PROGRAM High
VAR
	new : REAL := 0;
	change : REAL := 0;
END_VAR
VAR // added by the converter: edge detectors and wires of the graphical bodies
    _w1 : BOOL;
END_VAR

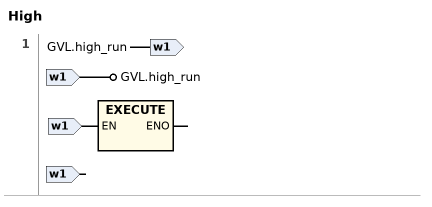
// NETWORK 1
_w1 := GVL.high_run;
GVL.high_run := NOT _w1;
IF _w1 THEN  END_IF

END_PROGRAM

(* stored: Version 1.1.0.1, ProductVersion 3.1.4024.12
   POU High: Id {ce067dc0-44d6-4633-ad05-d08be40dd68e}, SpecialFunc None *)
